TYPE XYZ_Point :
STRUCT
	X:LREAL;
	Y:LREAL;
	Z:LREAL;
END_STRUCT
END_TYPE

(* stored: Version 1.1.0.1, ProductVersion 3.1.4026.18
   DUT XYZ_Point: Id {c26f8907-94b5-4546-8eec-64d5e7e7672f} *)
